ADAPTER IFlushReq (* Adapter Interface *)
  (* Standard: 61499-1 *)
  (* Version 0.0, 6/23/2026, Schneider Electric *)
  PACKAGE SE.Nereda;
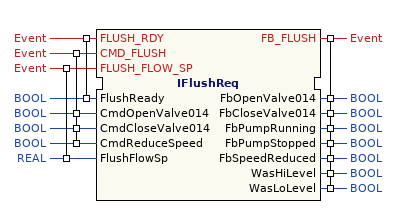
  EVENT_INPUT
    FLUSH_RDY WITH FlushReady;
    CMD_FLUSH WITH CmdOpenValve014, CmdCloseValve014, CmdReduceSpeed;
    FLUSH_FLOW_SP WITH FlushFlowSp;
  END_EVENT
  EVENT_OUTPUT
    FB_FLUSH WITH FbOpenValve014, FbCloseValve014, FbSpeedReduced, FbPumpRunning, FbPumpStopped, WasHiLevel, WasLoLevel;
  END_EVENT
  VAR_INPUT
    FlushReady : BOOL;
    CmdOpenValve014 : BOOL;
    CmdCloseValve014 : BOOL;
    CmdReduceSpeed : BOOL;
    FlushFlowSp : REAL;
  END_VAR
  VAR_OUTPUT
    FbOpenValve014 : BOOL;
    FbCloseValve014 : BOOL;
    FbPumpRunning : BOOL;
    FbPumpStopped : BOOL;
    FbSpeedReduced : BOOL;
    WasHiLevel : BOOL;
    WasLoLevel : BOOL;
  END_VAR
  SERVICE SOCKET/PLUG
    SEQUENCE request_confirm
      SOCKET.REQ(REQD) -> PLUG.REQ(REQD);
      PLUG.CMD_FLUSH(StartFlush) -> SOCKET.CMD_FLUSH(StartFlush);
    END_SEQUENCE
    SEQUENCE indication_response
      PLUG.IND(StopFlush) -> SOCKET.IND(StopFlush);
      SOCKET.RSP(RSPD) -> PLUG.RSP(RSPD);
    END_SEQUENCE
  END_SERVICE
END_ADAPTER
